FUNCTION_BLOCK TURNTABLE_MODEL (* Basic Function Block Type *)
  (* Standard: 61499-2 *)
  (* Version 0.3, 2009-09-15, JHC, Holobloc Inc, Changed transition priorities. *)
  (* Version 0.2, 2003-12-04, JHC, Rockwell Automation, Renamed for better indexing. *)
  (* Version 0.1, 2002-11-05, JHC, Rockwell Automation, Corrected missing ST element in Algorithm REQ. *)
  (* Version 0.0, 2000-05-30, JHC, Rockwell Automation *)
  PACKAGE fb.rt.Conveyer;
  IMPORT fb.datatype.*;
  IMPORT fb.rt.*;
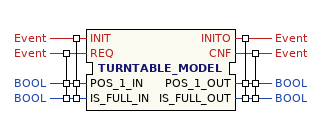
  EVENT_INPUT
    INIT WITH POS_1_IN, IS_FULL_IN; (* Initialization Request *)
    REQ WITH POS_1_IN, IS_FULL_IN; (* Normal Execution Request *)
  END_EVENT
  EVENT_OUTPUT
    INITO WITH POS_1_OUT, IS_FULL_OUT; (* Initialization Confirm *)
    CNF WITH POS_1_OUT, IS_FULL_OUT; (* Execution Confirmation *)
  END_EVENT
  VAR_INPUT
    POS_1_IN : BOOL;
    IS_FULL_IN : BOOL;
  END_VAR
  VAR_OUTPUT
    POS_1_OUT : BOOL;
    IS_FULL_OUT : BOOL;
  END_VAR
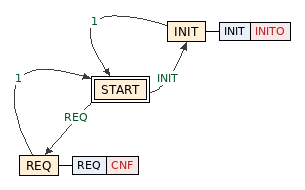
  EC_STATES
    START; (* Initial State *)
    INIT : INIT -> INITO; (* Initialization *)
    REQ : REQ -> CNF; (* Normal execution *)
  END_STATES
  EC_TRANSITIONS
    INIT TO START := 1;
    START TO REQ := REQ;
    START TO INIT := INIT;
    REQ TO START := 1;
  END_TRANSITIONS
  ALGORITHM INIT IN ST: (* Initialization algorithm *)
POS_1_OUT := TRUE;
IS_FULL_OUT := FALSE;
  END_ALGORITHM
  ALGORITHM REQ IN ST: (* Normally executed algorithm *)
POS_1_OUT := POS_1_IN;
IS_FULL_OUT := IS_FULL_IN;
  END_ALGORITHM
END_FUNCTION_BLOCK
